// TIA Portal V16 export
// export: Created 2021-09-08T12:44:32.20342Z, ExportSetting WithDefaults, DisplayName Totally Integrated Automation Portal, DisplayVersion V16 Update 3, DisplayName TIA Portal Version Control Interface, DisplayVersion V16 Update 2, DisplayName TIA Portal Openness, DisplayVersion V16 Update 3, DisplayName TIA Portal Teamcenter Gateway, DisplayVersion V16, DisplayName STEP 7 Professional, DisplayVersion V16 Update 3, DisplayName STEP 7 Safety, DisplayVersion V16, DisplayName WinCC Advanced, DisplayVersion V16 Update 3
VAR_GLOBAL   // PLC tag table "A10_DI"
   iDP101_Run AT %I2.0 : Bool;   // DP101 Робота
   iDP101_Fail AT %I2.1 : Bool;   // DP101 Аварія
   iDP502_Run AT %I2.2 : Bool;   // DP502 Робота
   iDP502_Fail AT %I2.3 : Bool;   // DP502 Аварія
   iDP501_Run AT %I2.4 : Bool;   // DP501 Робота
   iDP501_Fail AT %I2.5 : Bool;   // DP501 Аварія
   iDP801_Run AT %I2.6 : Bool;   // DP801 Робота
   iDP801_Fail AT %I2.7 : Bool;   // DP801 Аварія
   iDP802_Run AT %I3.0 : Bool;   // DP802 Робота
   iDP802_Fail AT %I3.1 : Bool;   // DP802 Аварія
   iDP803_Run AT %I3.2 : Bool;   // DP803 Робота
   iDP803_Fail AT %I3.3 : Bool;   // DP803 Аварія
   iDP1001_Run AT %I3.4 : Bool;   // DP1001 Робота
   iDP1001_Fail AT %I3.5 : Bool;   // DP1001 Аварія
   iUV1601_Fail AT %I3.6 : Bool;   // UV1601 Аварія
   "I3.7_Reserve" AT %I3.7 : Bool;   // Резерв
   iPS901 AT %I4.0 : Bool;   // Тиск на вході насоса зворотнього осмоса PS901
   iPS902 AT %I4.1 : Bool;   // Тиск перемеата зворотнього осмоса PS902
   iPS1301 AT %I4.2 : Bool;   // Тиск на вході насоса нанофільтрації PS1301
   iPS1302 AT %I4.3 : Bool;   // Тиск перемеата нанофільтрації PS1302
   iFL501 AT %I4.4 : Bool;   // Витрата повітря на промивку ультрафільтрації FL501
   iFL901 AT %I4.5 : Bool;   // Витрата рециклу зворотнього осмоса FL901
   iFL1301 AT %I4.6 : Bool;   // Витрата рециклу нанофільтрації FL1301
   iFM201 AT %I4.7 : Bool;   // Витрата вхідної води FM201
   iFM1201 AT %I5.0 : Bool;   // Витрата пермеату на споживоча FM1201
   iFM1701 AT %I5.1 : Bool;   // Витрата нанофільтрату на споживоча FM1701
   iFM1801 AT %I5.2 : Bool;   // Витрата стічних вод FM1801
   iFM501 AT %I5.3 : Bool;   // Витрата вхідної води UF FM501
   iFM502 AT %I5.4 : Bool;   // Витрата вхідної води UF FM502
   iFM901 AT %I5.5 : Bool;   // Витрата пермеату RO FM901
   iFM902 AT %I5.6 : Bool;   // Витрата концентрату RO FM902
   iFM1301 AT %I5.7 : Bool;   // Витрата пермеату NF FM1301
   iFM1302 AT %I6.0 : Bool;   // Витрата концентрату NF FM1302
   iDVA501_closed AT %I6.1 : Bool;   // Клапан DVA501 закрит
   iDVA501_open AT %I6.2 : Bool;   // Клапан DVA501 открит
   iDVA502_closed AT %I6.3 : Bool;   // Клапан DVA502 закрит
   iDVA502_open AT %I6.4 : Bool;   // Клапан DVA502 открит
   iDVA504_closed AT %I6.5 : Bool;   // Клапан DVA504 закрит
   iDVA504_open AT %I6.6 : Bool;   // Клапан DVA504 открит
   "I6.7_reserve" AT %I6.7 : Bool;   // Резерв
   iDVA505_closed AT %I7.0 : Bool;   // Клапан DVA505 закрит
   iDVA505_open AT %I7.1 : Bool;   // Клапан DVA505 открит
   iDVA506_closed AT %I7.2 : Bool;   // Клапан DVA506 закрит
   iDVA506_open AT %I7.3 : Bool;   // Клапан DVA506 открит
   iDVA507_closed AT %I7.4 : Bool;   // Клапан DVA507 закрит
   iDVA507_open AT %I7.5 : Bool;   // Клапан DVA507 открит
   iDVA508_closed AT %I7.6 : Bool;   // Клапан DVA508 закрит
   iDVA508_open AT %I7.7 : Bool;   // Клапан DVA508 открит
   iDVA509_closed AT %I8.0 : Bool;   // Клапан DVA509 закрит
   iDVA509_open AT %I8.1 : Bool;   // Клапан DVA509 открит
   iDVA511_closed AT %I8.2 : Bool;   // Клапан DVA511 закрит
   iDVA511_open AT %I8.3 : Bool;   // Клапан DVA511 открит
   iDVA512_closed AT %I8.4 : Bool;   // Клапан DVA512 закрит
   iDVA512_open AT %I8.5 : Bool;   // Клапан DVA512 открит
   iDVA513_closed AT %I8.6 : Bool;   // Клапан DVA513 закрит
   iDVA513_open AT %I8.7 : Bool;   // Клапан DVA513 открит
   iDVA514_closed AT %I9.0 : Bool;   // Клапан DVA514 закрит
   iDVA514_open AT %I9.1 : Bool;   // Клапан DVA514 открит
   iDVA515_closed AT %I9.2 : Bool;   // Клапан DVA515 закрит
   iDVA515_open AT %I9.3 : Bool;   // Клапан DVA515 открит
   iDVA516_closed AT %I9.4 : Bool;   // Клапан DVA516 закрит
   iDVA516_open AT %I9.5 : Bool;   // Клапан DVA516 открит
   iDVA1801_closed AT %I9.6 : Bool;   // Клапан DVA1801 закрит
   iDVA1801_open AT %I9.7 : Bool;   // Клапан DVA1801 открит
   iP3xx_Stop AT %I10.0 : Bool;   // P3xx Аварійне вимиканя
   iP901_Stop AT %I10.1 : Bool;   // P901 Аварійне вимиканя
   iP1301_Stop AT %I10.2 : Bool;   // P13xx Аварійне вимиканя
   iP12xx_Stop AT %I10.3 : Bool;   // P12xx Аварійне вимиканя
   iP15xx_Stop AT %I10.4 : Bool;   // P15xx Аварійне вимиканя
   iP7xx_Stop AT %I10.5 : Bool;   // P7xx Аварійне вимиканя
   iP2001_Stop AT %I10.6 : Bool;   // P2001 Аварійне вимиканя
   "I10.7_reserve" AT %I10.7 : Bool;   // Резерв
   "I11.0_reserve" AT %I11.0 : Bool;   // Резерв
   "I11.1_reserve" AT %I11.1 : Bool;   // Резерв
   "I11.2_reserve" AT %I11.2 : Bool;   // Резерв
   "I11.3_reserve" AT %I11.3 : Bool;   // Резерв
   "I11.4_reserve" AT %I11.4 : Bool;   // Резерв
   "I11.5_reserve" AT %I11.5 : Bool;   // Резерв
   "I11.6_reserve" AT %I11.6 : Bool;   // Резерв
   "I11.7_reserve" AT %I11.7 : Bool;   // Резерв
END_VAR
VAR_GLOBAL CONSTANT   // user constants
   "iDP-101_Run" : Int := 0;
   "iDP-101_Fail" : Int := 1;
   "iDP-502_Run" : Int := 2;
   "iDP-502_Fail" : Int := 3;
   "iDP-501_Run" : Int := 4;
   "iDP-501_Fail" : Int := 5;
   "iDP-801_Run" : Int := 6;
   "iDP-801_Fail" : Int := 7;
   "iDP-802_Run" : Int := 8;
   "iDP-802_Fail" : Int := 9;
   "iDP-803_Run" : Int := 10;
   "iDP-803_Fail" : Int := 11;
   "iDP-1001_Run" : Int := 12;
   "iDP-1001_Fail" : Int := 13;
   "iUV-1601_Fail" : Int := 14;
   "I3.7_res" : Int := 15;
   i_PS901 : Int := 16;
   i_PS902 : Int := 17;
   i_PS1301 : Int := 18;
   i_PS1302 : Int := 19;
   i_FL501 : Int := 20;
   i_FL901 : Int := 21;
   i_FL1301 : Int := 22;
   i_FM201 : Int := 23;
   i_FM1201 : Int := 24;
   i_FM1701 : Int := 25;
   i_FM1801 : Int := 26;
   i_FM501 : Int := 27;
   i_FM502 : Int := 28;
   i_FM901 : Int := 29;
   i_FM902 : Int := 30;
   i_FM1301 : Int := 31;
   i_FM1302 : Int := 32;
   "iDVA-501_closed" : Int := 33;
   "iDVA-501_open" : Int := 34;
   "iDVA-502_closed" : Int := 35;
   "iDVA-502_open" : Int := 36;
   "iDVA-504_closed" : Int := 37;
   "iDVA-504_open" : Int := 38;
   "I6.7_res" : Int := 39;
   "iDVA-505_closed" : Int := 40;
   "iDVA-505_open" : Int := 41;
   "iDVA-506_closed" : Int := 42;
   "iDVA-506_open" : Int := 43;
   "iDVA-507_closed" : Int := 44;
   "iDVA-507_open" : Int := 45;
   "iDVA-508_closed" : Int := 46;
   "iDVA-508_open" : Int := 47;
   "iDVA-509_closed" : Int := 48;
   "iDVA-509_open" : Int := 49;
   "iDVA-511_closed" : Int := 50;
   "iDVA-511_open" : Int := 51;
   "iDVA-512_closed" : Int := 52;
   "iDVA-512_open" : Int := 53;
   "iDVA-513_closed" : Int := 54;
   "iDVA-513_open" : Int := 55;
   "iDVA-514_closed" : Int := 56;
   "iDVA-514_open" : Int := 57;
   "iDVA-515_closed" : Int := 58;
   "iDVA-515_open" : Int := 59;
   "iDVA-516_closed" : Int := 60;
   "iDVA-516_open" : Int := 61;
   "iDVA-1801_closed" : Int := 62;
   "iDVA-1801_open" : Int := 63;
   "iP-3xx_Stop" : Int := 64;
   "iP-901_Stop" : Int := 65;
   "iP-1301_Stop" : Int := 66;
   "iP-12xx_Stop" : Int := 67;
   "iP-15xx_Stop" : Int := 68;
   "iP-7xx_Stop" : Int := 69;
   "iP-2001_Stop" : Int := 70;
   "I10.7_res" : Int := 71;
   "I11.0_res" : Int := 72;
   "I11.1_res" : Int := 73;
   "I11.2_res" : Int := 74;
   "I11.3_res" : Int := 75;
   "I11.4_res" : Int := 76;
   "I11.5_res" : Int := 77;
   "I11.6_res" : Int := 78;
   "I11.7_res" : Int := 79;
END_VAR
